PROGRAM Q5
VAR
	i : INT := 0;
 	output : BOOL := FALSE;
END_VAR

(*
init:
	i is an INT init to 0
	output is a BOOL init to false

1:
	0 is assigned to i
	
	i == 0
	
2:
	if i > 0, not goto label default
	
	i is not > 0, therefore goto -> default:
	
3:
	TRUE is assigned to output
	
	not executed as it was jumped by the goto label

4:
	label default, no functionality
	
	no functionality, return
	
end:
	output has value FALSE at the end of execution

*)

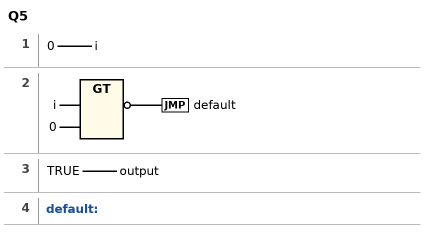
// NETWORK 1
i := 0;

// NETWORK 2
IF NOT (i > 0) THEN JMP default; END_IF

// NETWORK 3
output := TRUE;

// NETWORK 4
default: ;

END_PROGRAM

(* stored: Version 1.1.0.1, ProductVersion 3.1.4024.12
   POU Q5: Id {beae2521-7db7-4f96-b8d9-e0c6834ca460}, SpecialFunc None *)
